# EPICS substitutions: iocBoot/iocSolaris/motorSim.substitutions
file "$(MOTOR)/db/basic_asyn_motor.db"
{
pattern
{P,     N,  M,      DTYP,            PORT, ADDR,  DESC,          EGU,      DIR,  VELO,  VBAS,  ACCL,  BDST,  BVEL,  BACC,  MRES,  PREC,  DHLM,  DLLM,  INIT}
{CARS:,  1,  "m$(N)",  "asynMotor",  motorSim1,  0,  "motor $(N)",  degrees,  Pos,  1,     .1,    .2,    0,     1,     .2,    0.01,  5,     100,   -100,  ""}
{CARS:,  2,  "m$(N)",  "asynMotor",  motorSim1,  1,  "motor $(N)",  degrees,  Pos,  1,     .1,    .2,    0,     1,     .2,    0.01,  5,     100,   -100,  ""}
{CARS:,  3,  "m$(N)",  "asynMotor",  motorSim1,  2,  "motor $(N)",  degrees,  Pos,  1,     .1,    .2,    0,     1,     .2,    0.01,  5,     100,   -100,  ""}
{CARS:,  4,  "m$(N)",  "asynMotor",  motorSim1,  3,  "motor $(N)",  degrees,  Pos,  1,     .1,    .2,    0,     1,     .2,    0.01,  5,     100,   -100,  ""}
{CARS:,  5,  "m$(N)",  "asynMotor",  motorSim1,  4,  "motor $(N)",  degrees,  Pos,  1,     .1,    .2,    0,     1,     .2,    0.01,  5,     100,   -100,  ""}
{CARS:,  6,  "m$(N)",  "asynMotor",  motorSim1,  5,  "motor $(N)",  degrees,  Pos,  1,     .1,    .2,    0,     1,     .2,    0.01,  5,     100,   -100,  ""}
{CARS:,  7,  "m$(N)",  "asynMotor",  motorSim1,  6,  "motor $(N)",  degrees,  Pos,  1,     .1,    .2,    0,     1,     .2,    0.01,  5,     100,   -100,  ""}
{CARS:,  8,  "m$(N)",  "asynMotor",  motorSim1,  7,  "motor $(N)",  degrees,  Pos,  1,     .1,    .2,    0,     1,     .2,    0.01,  5,     100,   -100,  ""}
}
